FUNCTION FC_Variance : REAL
VAR_INPUT
a: ARRAY [1..10] OF REAL;
END_VAR
VAR
b:REAL;
test:BOOL;
ii1:INT;
c:REAL;
d:real;
END_VAR

test:=FALSE;
FOR ii1:=1 TO 10 BY 1 DO
	IF a[ii1]=0 THEN
		test:=TRUE;
	END_IF
END_FOR
IF test THEN
	FC_Variance:=0;
ELSE
	b:=0;
	//FOR ii1:=1 TO 10 BY 1 DO
	//	b:=b+a[ii1];
	//END_FOR	
	c:=b/10;	
	d:=0;
	FOR ii1:=1 TO 10 BY 1 DO
		d:=d+(c-a[ii1])*(c-a[ii1]);
	END_FOR
	FC_Variance:=d/10;
END_IF

END_FUNCTION

(* stored: Version 1.1.0.1, ProductVersion 3.1.4024.9
   POU FC_Variance: Id {bac0c29f-c1f4-4573-9e4c-b4971535437f}, SpecialFunc None *)
